FUNCTION_BLOCK AX_F_TRIG (* Boolean falling edge detection *)
  (* Standard: 61499-1 Annex A; Description: Copyright (c) 2017 fortiss GmbH, HR Agrartechnik GmbH This program and the accompanying materials are made available under the terms of the Eclipse Public License 2.0 which is available at https://www.eclipse.org/legal/epl-2.0/ SPDX-License-Identifier: EPL-2.0 *)
  (* Version 3.0, 2025-04-14, Patrick Aigner, changed package *)
  (* Version 1.0, 2017-09-22, Alois Zoitl, fortiss GmbH, initial API and implementation and/or initial documentation *)
  PACKAGE adapter::events::unidirectional;
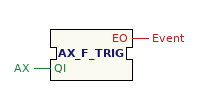
  EVENT_OUTPUT
    EO; (* confirmation that an falling edge was detected *)
  END_EVENT
  SOCKETS
    QI : adapter::types::unidirectional::AX; (* value to check for a falling edge *)
  END_SOCKETS
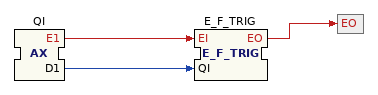
  FBS
    E_F_TRIG : iec61499::events::E_F_TRIG;
  END_FBS
  EVENT_CONNECTIONS
    QI.E1 TO E_F_TRIG.EI;
    E_F_TRIG.EO TO EO;
  END_CONNECTIONS
  DATA_CONNECTIONS
    QI.D1 TO E_F_TRIG.QI;
  END_CONNECTIONS
END_FUNCTION_BLOCK
